Universal Robots PolyScope program: SyntaxError.urp

ProgramRoot directory=/home/ur/ursim-3.1/programs/SyntaxError; kinematics=(a=[0, -0.612, -0.5723, 0, 0, 0], d=[0.1273, 0, 0, 0.16394, 0.1157, 0.0922], alpha=[1.5708, 0, 0, 1.5708, -1.5708, 0], deltaTheta=[0, 0, 0, 0, 0, 0], status=notInitialized); lastSavedInVersion=(project__name=Polyscope, major__version=3, minor__version=1, svn__revision=16916, build__date=Feb 06 2015, 15:15:00); name=SyntaxError; programVersion=(project__name=PolyScope, major__version=1, minor__version=8, svn__revision=11281, build__date=Aug 07 2013, 11:50:39); robotEnvironmentFileName=default; serialNumberRobot=2014350001
  MainProgram cartesianAcceleration=1.2; cartesianSpeed=0.25; jointAcceleration=1.3962634015954636; jointSpeed=1.0471975511965976; sharedProcessMoveBlendRadius=0.025; motionType=JOINT_SPACE
    Move cartesianAcceleration=1.2; cartesianSpeed=0.25; jointAcceleration=1.3962634015954636; jointSpeed=1.0471975511965976; sharedProcessMoveBlendRadius=0.025; motionType=JOINT_SPACE
      Waypoint blendRadius=0.05; cartesianAcceleration=1.2; cartesianSpeed=0.25; jointAcceleration=1.3962634015954636; jointSpeed=1.0471975511965976; nextMotionTime=2.0; stoppoint=true; useSharedBlendParameter=true; useSharedParameters=true; outputFlangePose=(pos=(x=-0.12012816514413963, y=-0.43226726300653034, z=0.32303919034329), rot=(x=-0.001221364921157579, y=3.1162765249936863, z=0.03889192061104669)); position=TCP in base x=-180.005 y=-609.524 z=488.915 mm, rx=-0.0012 ry=3.1163 rz=0.0389 rad; joints [-91.713, -85.307, -110.221, -75.944, 91.392, -1.776] deg; positionType=FIXED_POSITION; waypointPoseInFeatureCoordinates=(pos=(x=-0.18000518706228327, y=-0.609523887683218, z=0.48891530024105245), rot=(x=-0.0012213649211588729, y=3.1162765249936863, z=0.038891920611046675)); name=路点_1
      Assignment expr=get_target_tcp_pose(); operatorValueType=INTEGER; valueSource=EXPRESSION
      Assignment expr=get_target_tcp_pose(); operatorValueType=INTEGER; valueSource=EXPRESSION
      Assignment expr=pose_add(ExpressionVariableNode,p[0,0,0.1,0,0,0]); operatorValueType=INTEGER; valueSource=EXPRESSION
      Waypoint blendRadius=0.05; cartesianAcceleration=1.2; cartesianSpeed=0.25; jointAcceleration=1.3962634015954636; jointSpeed=1.0471975511965976; nextMotionTime=2.0; stoppoint=true; useSharedBlendParameter=true; useSharedParameters=true; positionType=VARIABLE_POSITION; name=var_3
      Waypoint blendRadius=0.05; cartesianAcceleration=1.2; cartesianSpeed=0.25; jointAcceleration=1.3962634015954636; jointSpeed=1.0471975511965976; nextMotionTime=2.0; stoppoint=true; useSharedBlendParameter=true; useSharedParameters=true; positionType=VARIABLE_POSITION; name=var_3
